FUNCTION F_GetValueString : STRING
VAR_INPUT
	Symbol : ANY;
END_VAR

VAR
	ubuff  : ULINT;
	sibuff : SINT;
	ibuff  : INT;
	dibuff : DINT;
	libuff : LINT;
	rbuff  : REAL;
    lrbuff : LREAL;
	sbuff  : STRING(255);
	wsbuff : WSTRING(255);
	x	   : INT; // loop var for STRING and WSTRING
END_VAR

F_GetValueString := '';
CASE Symbol.TypeClass OF
	__SYSTEM.TYPE_CLASS.TYPE_BOOL:
		memcpy(ADR(ubuff), Symbol.pValue, Symbol.diSize);
		F_GetValueString := TO_STRING(TO_BOOL(TO_LREAL(ubuff)));

	__SYSTEM.TYPE_CLASS.TYPE_BYTE, __SYSTEM.TYPE_CLASS.TYPE_USINT, __SYSTEM.TYPE_CLASS.TYPE_WORD, __SYSTEM.TYPE_CLASS.TYPE_UINT, __SYSTEM.TYPE_CLASS.TYPE_DWORD, __SYSTEM.TYPE_CLASS.TYPE_UDINT, __SYSTEM.TYPE_CLASS.TYPE_LWORD, __SYSTEM.TYPE_CLASS.TYPE_ULINT:
		memcpy(ADR(ubuff), Symbol.pValue, Symbol.diSize);
		F_GetValueString := LREAL_TO_FMTSTR(TO_LREAL(ubuff), 0, FALSE);

	__SYSTEM.TYPE_CLASS.TYPE_SINT:
		memcpy(ADR(sibuff), Symbol.pValue, Symbol.diSize);
		F_GetValueString := LREAL_TO_FMTSTR(TO_LREAL(sibuff), 0, FALSE);

	__SYSTEM.TYPE_CLASS.TYPE_INT:
		memcpy(ADR(ibuff), Symbol.pValue, Symbol.diSize);
		F_GetValueString := LREAL_TO_FMTSTR(TO_LREAL(ibuff), 0, FALSE);

	__SYSTEM.TYPE_CLASS.TYPE_DINT:
		memcpy(ADR(dibuff), Symbol.pValue, Symbol.diSize);
		F_GetValueString := LREAL_TO_FMTSTR(TO_LREAL(dibuff), 0, FALSE);

	__SYSTEM.TYPE_CLASS.TYPE_LINT:
		memcpy(ADR(libuff), Symbol.pValue, Symbol.diSize);
		F_GetValueString := LREAL_TO_FMTSTR(TO_LREAL(libuff), 0, FALSE);

	__SYSTEM.TYPE_CLASS.TYPE_REAL, __SYSTEM.TYPE_CLASS.TYPE_LREAL:
		IF Symbol.TypeClass = __SYSTEM.TYPE_CLASS.TYPE_REAL THEN
			memcpy(ADR(rbuff), Symbol.pValue, Symbol.diSize);
			F_GetValueString := LREAL_TO_FMTSTR(TO_LREAL(rbuff), 5, TRUE);
		ELSIF Symbol.TypeClass = __SYSTEM.TYPE_CLASS.TYPE_LREAL THEN
			memcpy(ADR(lrbuff), Symbol.pValue, Symbol.diSize);
			F_GetValueString := LREAL_TO_FMTSTR(TO_LREAL(lrbuff), 5, TRUE);
		END_IF

	__SYSTEM.TYPE_CLASS.TYPE_STRING, __SYSTEM.TYPE_CLASS.TYPE_WSTRING:
		IF Symbol.TypeClass = __SYSTEM.TYPE_CLASS.TYPE_STRING THEN
			MEMCPY(ADR(sbuff), Symbol.pValue, MIN(SIZEOF(sbuff), TO_UDINT(Symbol.diSize)));
		ELSIF Symbol.TypeClass = __SYSTEM.TYPE_CLASS.TYPE_WSTRING THEN
			MEMCPY(ADR(wsbuff), Symbol.pValue, MIN(SIZEOF(wsbuff), TO_UDINT(Symbol.diSize)));
			WSTRING_TO_STRING2(ADR(sbuff), ADR(wsbuff), SIZEOF(sbuff));
		END_IF

		F_GetValueString := sbuff;
END_CASE

END_FUNCTION

(* stored: Version 1.1.0.1
   POU F_GetValueString: Id {d92f83d0-a528-4290-b20f-eeb6abd04e6a}, SpecialFunc None *)
